TYPE aT_Tank :
STRUCT
	HI: BOOL;
	LO: BOOL;
	Level: REAL;
END_STRUCT
END_TYPE

(* stored: Version 1.1.0.1, ProductVersion 3.1.4024.4
   DUT aT_Tank: Id {5592f321-3899-4157-9126-624a772cec25} *)
